FUNCTION_BLOCK FB_KUKA_MAIN
VAR_INPUT
END_VAR
VAR_OUTPUT
END_VAR
VAR
		JobRun 			:  BOOL := FALSE;
		bResetOUT		: BOOL := FALSE;
		bJob_InProcess	: BOOL := FALSE;
		iRackLocation: INT;
		Timer1			:	TON;
		
END_VAR

//If Soft EStop is pressed, turn off 1027 ~ 1034
IF IO_KUKA.KR_Estop OR NOT IO_control.bEstop OR IO_KUKA.bAlarm_stop = FALSE THEN		
	IO_control.bMove_enable := IO_control.bDrive_off := IO_control.bIO_Act := IO_control.bExt_start:=
	IO_control.bConf_msg := IO_control.bDrive_on := IO_HMI.bMove_enable := IO_HMI.bDrive_off := IO_HMI.bIO_Act := IO_HMI.bExt_start := IO_HMI.bConf_msg := IO_HMI.bDrive_on := FALSE;
END_IF

//Idle monitor all prog byte x running 	
IF IO_KUKA.PLC_I_D1 = 1 AND IO_KUKA.PLC_I_D2 = 0 THEN
	IO_KUKA.Idle := TRUE;
ELSE
	IO_KUKA.Idle := FALSE;
END_IF

//Online monitor T!/EXT mode
IF IO_KUKA.bEXT_mode THEN
	IO_KUKA.KROnline := TRUE;
	//IO.sKUKA_Online_val := '1';
ELSE
	IO_KUKA.KROnline := FALSE;
	//IO.sKUKA_Online_val := '0';
END_IF

//KUKA standby (ext mode) ---pro_act monitoring
IF IO_KUKA.bPro_act THEN
	IO_KUKA.KR_OnStandby := TRUE;
ELSE
	IO_KUKA.KR_OnStandby := FALSE;
END_IF


Timer1(IN:= IO_KUKA.bBin_pickup_InProcess  , PT:= T#5S);

IF IO_KUKA.KR_OnStandby AND IO_Conveyor.bKUKA_Job_Start THEN
	CASE IO.iRackLocation OF
		
		//initilize
		0:	JobRun := FALSE;
			IO_Conveyor.bPickup_Done := FALSE ;
			//IO_Conveyor.bKUKA_Job_Start := FALSE;
		
			
	(*================================ RackA : Pos1 =======================================*)	
		//203
		1:	IF NOT JobRun THEN
				IO_control.bRA_pos1 := TRUE;
			END_IF
		
			IF IO_KUKA.bBin_pickup_InProcess = TRUE THEN
				JobRun := TRUE;
			END_IF
			
			IF JobRun THEN
				IF IO_KUKA.bBin_pickup_InProcess = FALSE THEN
					IO_Conveyor.bPickup_Done := TRUE;
					bResetOUT := TRUE;
					IF IO_KUKA.bRA_pos1_InProcess = FALSE THEN
						IO_Conveyor.bKUKA_Job_Done := TRUE;
						IO.iRackLocation := 0;
					END_IF
				END_IF
			END_IF
	
	
	(*================================ RackA : Pos2 =======================================*)			
		2:	IF NOT JobRun THEN
				IO_control.bRA_pos2 := TRUE;
			END_IF
		
			IF IO_KUKA.bBin_pickup_InProcess = TRUE THEN
				JobRun := TRUE;
//				IF Timer1.Q THEN
//					bResetOUT := TRUE;
//				END_IF
			END_IF
			
			IF JobRun THEN
				IF IO_KUKA.bBin_pickup_InProcess = FALSE THEN
					IO_Conveyor.bPickup_Done := TRUE;
					bResetOUT := TRUE;
					IF IO_KUKA.bRA_pos2_InProcess = FALSE THEN
						IO_Conveyor.bKUKA_Job_Done := TRUE;
						IO.iRackLocation := 0;
					END_IF
				END_IF
			END_IF
	

	(*================================ RackA : Pos3 =======================================*)			
		3:	IF NOT JobRun THEN
				IO_control.bRA_pos3 := TRUE;
			END_IF
		
			IF IO_KUKA.bBin_pickup_InProcess = TRUE THEN
				JobRun := TRUE;
				//IO_control.bRA_pos3 := FALSE;
			END_IF
			
			IF JobRun THEN
				IF IO_KUKA.bBin_pickup_InProcess = FALSE THEN
					IO_Conveyor.bPickup_Done := TRUE;
					bResetOUT := TRUE;
					IF IO_KUKA.bRA_pos3_InProcess = FALSE THEN
						IO_Conveyor.bKUKA_Job_Done := TRUE;
						IO.iRackLocation := 0;
					END_IF
				END_IF
			END_IF
	
	
	(*================================ RackA : Pos4 =======================================*)				
		4:	IF NOT JobRun THEN
				IO_control.bRA_pos4 := TRUE;
			END_IF
		
			IF IO_KUKA.bBin_pickup_InProcess = TRUE THEN
				JobRun := TRUE;
				//IO_control.bRA_pos4 := FALSE;
			END_IF
			
			IF JobRun THEN
				IF IO_KUKA.bBin_pickup_InProcess = FALSE THEN
					IO_Conveyor.bPickup_Done := TRUE;
					bResetOUT := TRUE;
					IF IO_KUKA.bRA_pos4_InProcess = FALSE THEN
						IO_Conveyor.bKUKA_Job_Done := TRUE;
						IO.iRackLocation := 0;
					END_IF
				END_IF
			END_IF
	

	(*================================ RackA : Pos5 =======================================*)			
		5:	IF NOT JobRun THEN
				IO_control.bRA_pos5 := TRUE;
			END_IF
		
			IF IO_KUKA.bBin_pickup_InProcess = TRUE THEN
				JobRun := TRUE;
				//IO_control.bRA_pos5 := FALSE;
			END_IF
			
			IF JobRun THEN
				IF IO_KUKA.bBin_pickup_InProcess = FALSE THEN
					IO_Conveyor.bPickup_Done := TRUE;
					bResetOUT := TRUE;
					IF IO_KUKA.bRA_pos5_InProcess = FALSE THEN
						IO_Conveyor.bKUKA_Job_Done := TRUE;
						IO.iRackLocation := 0;
					END_IF
				END_IF
			END_IF
	

	(*================================ RackA : Pos6 =======================================*)				
		6:	IF NOT JobRun THEN
				IO_control.bRA_pos6 := TRUE;
			END_IF
		
			IF IO_KUKA.bBin_pickup_InProcess = TRUE THEN
				JobRun := TRUE;
				//IO_control.bRA_pos6 := FALSE;
			END_IF
			
			IF JobRun THEN
				IF IO_KUKA.bBin_pickup_InProcess = FALSE THEN
					IO_Conveyor.bPickup_Done := TRUE;
					bResetOUT := TRUE;
					IF IO_KUKA.bRA_pos6_InProcess = FALSE THEN
						IO_Conveyor.bKUKA_Job_Done := TRUE;
						IO.iRackLocation := 0;
					END_IF
				END_IF
			END_IF
	

	(*================================ RackB : Pos7 =======================================*)						
		7:	IF NOT JobRun THEN
				IO_control.bRB_pos7 := TRUE;
			END_IF
		
			IF IO_KUKA.bBin_pickup_InProcess = TRUE THEN
				JobRun := TRUE;
				//IO_control.bRB_pos7 := FALSE;
			END_IF
			
			IF JobRun THEN
				IF IO_KUKA.bBin_pickup_InProcess = FALSE THEN
					IO_Conveyor.bPickup_Done := TRUE;
					bResetOUT := TRUE;
					IF IO_KUKA.bRB_pos7_InProcess = FALSE THEN
						IO_Conveyor.bKUKA_Job_Done := TRUE;
						IO.iRackLocation := 0;
					END_IF
				END_IF
			END_IF
	

	(*================================ RackB : Pos8 =======================================*)		
		8:	IF NOT JobRun THEN
				IO_control.bRB_pos8 := TRUE;
			END_IF
		
			IF IO_KUKA.bBin_pickup_InProcess = TRUE THEN
				JobRun := TRUE;
				//IO_control.bRB_pos8 := FALSE;
			END_IF
			
			IF JobRun THEN
				IF IO_KUKA.bBin_pickup_InProcess = FALSE THEN
					IO_Conveyor.bPickup_Done := TRUE;
					bResetOUT := TRUE;
					IF IO_KUKA.bRB_pos8_InProcess = FALSE THEN
						IO_Conveyor.bKUKA_Job_Done := TRUE;
						IO.iRackLocation := 0;
					END_IF
				END_IF
			END_IF
	

	(*================================ RackB : Pos9 =======================================*)			
		9:	IF NOT JobRun THEN
				IO_control.bRB_pos9 := TRUE;
			END_IF
		
			IF IO_KUKA.bBin_pickup_InProcess = TRUE THEN
				JobRun := TRUE;
			//	IO_control.bRB_pos9 := FALSE;
			END_IF
			
			IF JobRun THEN
				IF IO_KUKA.bBin_pickup_InProcess = FALSE THEN
					IO_Conveyor.bPickup_Done := TRUE;
					bResetOUT := TRUE;
					IF IO_KUKA.bRB_pos9_InProcess = FALSE THEN
						IO_Conveyor.bKUKA_Job_Done := TRUE;
						IO.iRackLocation := 0;
					END_IF
				END_IF
			END_IF
	

	(*================================ RackB : Pos10 =======================================*)		
		10:	IF NOT JobRun THEN
				IO_control.bRB_pos10 := TRUE;
			END_IF
		
			IF IO_KUKA.bBin_pickup_InProcess = TRUE THEN
				JobRun := TRUE;
				//IO_control.bRB_pos10 := FALSE;
			END_IF
			
			IF JobRun THEN
				IF IO_KUKA.bBin_pickup_InProcess = FALSE THEN
					IO_Conveyor.bPickup_Done := TRUE;
					bResetOUT := TRUE;
					IF IO_KUKA.bRB_pos10_InProcess = FALSE THEN
						IO_Conveyor.bKUKA_Job_Done := TRUE;
						IO.iRackLocation := 0;
					END_IF
				END_IF
			END_IF
	

	(*================================ RackB : Pos11 =======================================*)			
		11:	IF NOT JobRun THEN
				IO_control.bRB_pos11 := TRUE;
			END_IF
		
			IF IO_KUKA.bBin_pickup_InProcess = TRUE THEN
				JobRun := TRUE;
				//IO_control.bRB_pos11 := FALSE;
			END_IF
			
			IF JobRun THEN
				IF IO_KUKA.bBin_pickup_InProcess = FALSE THEN
					IO_Conveyor.bPickup_Done := TRUE;
					bResetOUT := TRUE;
					IF IO_KUKA.bRB_pos11_InProcess = FALSE THEN
						IO_Conveyor.bKUKA_Job_Done := TRUE;
						IO.iRackLocation := 0;
					END_IF
				END_IF
			END_IF
	

	(*================================ RackB : Pos12 =======================================*)		
		12:	IF NOT JobRun THEN
				IO_control.bRB_pos12 := TRUE;
			END_IF
		
			IF IO_KUKA.bBin_pickup_InProcess = TRUE THEN
				JobRun := TRUE;
			//	IO_control.bRB_pos12 := FALSE;
			END_IF
			
			IF JobRun THEN
				IF IO_KUKA.bBin_pickup_InProcess = FALSE THEN
					IO_Conveyor.bPickup_Done := TRUE;
					bResetOUT := TRUE;
					IF IO_KUKA.bRB_pos12_InProcess = FALSE THEN
						IO_Conveyor.bKUKA_Job_Done := TRUE;
						IO.iRackLocation := 0;
					END_IF
				END_IF
			END_IF
	

	(*================================ RackC : Pos13 =======================================*)		
		13:	IF NOT JobRun THEN
				IO_control.bRC_pos13 := TRUE;
			END_IF
		
			IF IO_KUKA.bBin_pickup_InProcess = TRUE THEN
				JobRun := TRUE;
				//IO_control.bRC_pos13 := FALSE;
			END_IF
			
			IF JobRun THEN
				IF IO_KUKA.bBin_pickup_InProcess = FALSE THEN
					IO_Conveyor.bPickup_Done := TRUE;
					bResetOUT := TRUE;
					IF IO_KUKA.bRC_pos13_InProcess = FALSE THEN
						IO_Conveyor.bKUKA_Job_Done := TRUE;
						IO.iRackLocation := 0;
					END_IF
				END_IF
			END_IF	
	

	(*================================ RackC : Pos14 =======================================*)		
		14:	IF NOT JobRun THEN
				IO_control.bRC_pos14 := TRUE;
			END_IF
		
			IF IO_KUKA.bBin_pickup_InProcess = TRUE THEN
				JobRun := TRUE;
				//IO_control.bRC_pos14 := FALSE;
			END_IF
			
			IF JobRun THEN
				IF IO_KUKA.bBin_pickup_InProcess = FALSE THEN
					IO_Conveyor.bPickup_Done := TRUE;
					bResetOUT := TRUE;
					IF IO_KUKA.bRC_pos14_InProcess = FALSE THEN
						IO_Conveyor.bKUKA_Job_Done := TRUE;
						IO.iRackLocation := 0;
					END_IF
				END_IF
			END_IF			
	

	(*================================ RackC : Pos15 =======================================*)		
		15:	IF NOT JobRun THEN
				IO_control.bRC_pos15 := TRUE;
			END_IF
		
			IF IO_KUKA.bBin_pickup_InProcess = TRUE THEN
				JobRun := TRUE;
				//IO_control.bRC_pos15 := FALSE;
			END_IF
			
			IF JobRun THEN
				IF IO_KUKA.bBin_pickup_InProcess = FALSE THEN
					IO_Conveyor.bPickup_Done := TRUE;
					bResetOUT := TRUE;
					IF IO_KUKA.bRC_pos15_InProcess = FALSE THEN
						IO_Conveyor.bKUKA_Job_Done := TRUE;
						IO.iRackLocation := 0;
					END_IF
				END_IF
			END_IF	

			
	(*================================ RackC : Pos16 =======================================*)
		16:	IF NOT JobRun THEN
				IO_control.bRC_pos16 := TRUE;
			END_IF
		
			IF IO_KUKA.bBin_pickup_InProcess = TRUE THEN
				JobRun := TRUE;
				//IO_control.bRC_pos16 := FALSE;
			END_IF
			
			IF JobRun THEN
				IF IO_KUKA.bBin_pickup_InProcess = FALSE THEN
					IO_Conveyor.bPickup_Done := TRUE;
					bResetOUT := TRUE;
					IF IO_KUKA.bRC_pos16_InProcess = FALSE THEN
						IO_Conveyor.bKUKA_Job_Done := TRUE;
						IO.iRackLocation := 0;
					END_IF
				END_IF
			END_IF	
			
	(*================================ RackC : Pos17 =======================================*)
		17:	IF NOT JobRun THEN
				IO_control.bRC_pos17 := TRUE;
			END_IF
		
			IF IO_KUKA.bBin_pickup_InProcess = TRUE THEN
				JobRun := TRUE;
			//	IO_control.bRC_pos17 := FALSE;
			END_IF
			
			IF JobRun THEN
				IF IO_KUKA.bBin_pickup_InProcess = FALSE THEN
					IO_Conveyor.bPickup_Done := TRUE;
					bResetOUT := TRUE;
					IF IO_KUKA.bRC_pos17_InProcess = FALSE THEN
						IO_Conveyor.bKUKA_Job_Done := TRUE;
						IO.iRackLocation := 0;
					END_IF
				END_IF
			END_IF		
	

	(*================================ RackC : Pos18 =======================================*)	
		18:	IF NOT JobRun THEN
				IO_control.bRC_pos18 := TRUE;
			END_IF
		
			IF IO_KUKA.bBin_pickup_InProcess = TRUE THEN
				JobRun := TRUE;
			//	IO_control.bRC_pos18 := FALSE;
			END_IF
			
			IF JobRun THEN
				IF IO_KUKA.bBin_pickup_InProcess = FALSE THEN
					IO_Conveyor.bPickup_Done := TRUE;
					bResetOUT := TRUE;
					IF IO_KUKA.bRC_pos18_InProcess = FALSE THEN
						IO_Conveyor.bKUKA_Job_Done := TRUE;
						IO.iRackLocation := 0;
					END_IF
				END_IF
			END_IF	

	END_CASE
END_IF

IF bResetOUT THEN
	//IO_KUKA.PLC_O_D1 :=  1;
	IO_control.bRA_pos1 := IO_control.bRA_pos2 := IO_control.bRA_pos3 := IO_control.bRA_pos4 := IO_control.bRA_pos5 := IO_control.bRA_pos6 := IO_control.bRB_pos7 := IO_control.bRB_pos8 := IO_control.bRB_pos9 := IO_control.bRB_pos10 := IO_control.bRB_pos11 := IO_control.bRB_pos12 := IO_control.bRC_pos13 := IO_control.bRC_pos14 := IO_control.bRC_pos15 := IO_control.bRC_pos16 := IO_control.bRC_pos17 := IO_control.bRC_pos18 := FALSE;
	bResetOUT := FALSE;
END_IF

END_FUNCTION_BLOCK

(* stored: Version 1.1.0.1, ProductVersion 3.1.4024.12
   POU FB_KUKA_MAIN: Id {e8ab190c-a631-4882-8a93-6516c2fdb37c}, SpecialFunc None *)
